ABB RobotStudio station: 00_Proyecto_RI_Irene_Perdiguero.rspag

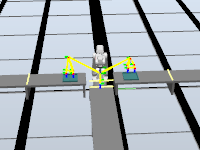
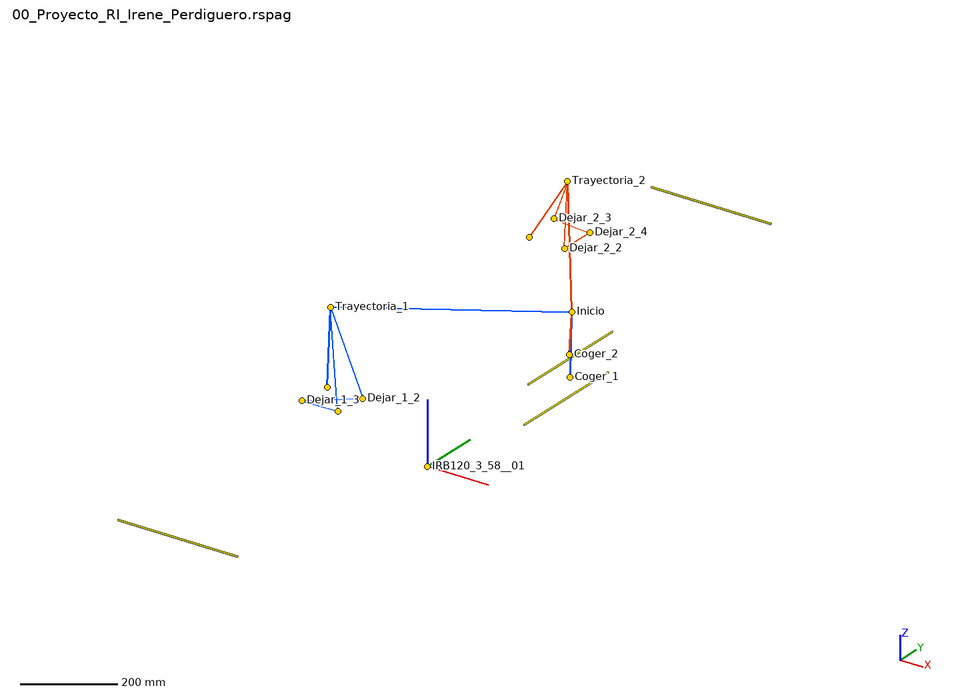
[picture v1: parts stored in the station drawn from their meshes, with robot base, taught points and paths (robot models come from the ABB library and are not in the file)]
--- station ---
Station 00_Proyecto_RI_Irene_Perdiguero (saved by RobotStudio 21.2.9526.0)
Controller Controlador1
  mechanical unit ROB_1: IRB120_3_58__01, 6 joints, base frame (0, 0, 0) mm
Layout (positions relative to the parent item):
  - IRB120_3_58__01 [mechanism, from Robots\IRB120_3_58_G_01.rslib] at (0, 0, 0) mm; joint values [-0.05, 0.292, -0.2841, -0.0016, 1.5947, -0.05] (rad or m)
  - Ventosa [mechanism, from Libraries\Ventosa.rslib] at (377.49, -19, 544.24) mm, rotated rx 180 ry -1.82 rz -180 deg
  - Producto_1 [part] at (808.06, -356.02, 0) mm, size 40 x 40 x 100 mm
  - Producto_2 [part] at (939.96, 363, 0) mm, size 40 x 39.4 x 150 mm
  - Cinta [smart component]
      signals: DI MARCHA, DI COGER_1, DI COGER_2, DI DEJAR_1, DI DEJAR_2, DO PRODUCTO_1, DO PRODUCTO_2
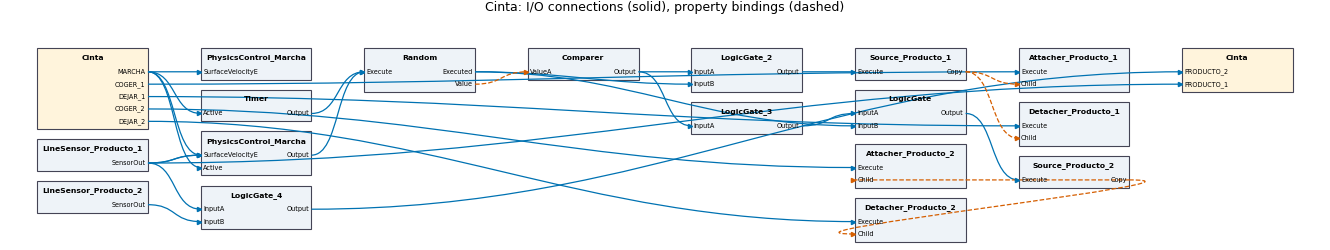
      connections:
        Cinta.MARCHA -> PhysicsControl_Marcha.SurfaceVelocityEnabled
        Cinta.MARCHA -> Timer.Active
        Timer.Output -> Random.Execute
        Comparer.Output -> LogicGate_2.InputA
        Comparer.Output -> LogicGate_3.InputA
        LogicGate_3.Output -> LogicGate.InputA
        Random.Executed -> LogicGate_2.InputB
        Random.Executed -> LogicGate.InputB
        LogicGate.Output -> Source_Producto_2.Execute
        LogicGate_2.Output -> Source_Producto_1.Execute
        LineSensor_Producto_1.SensorOut -> PhysicsControl_Paro.SurfaceVelocityEnabled
        LineSensor_Producto_1.SensorOut -> LogicGate_4.InputA
        LineSensor_Producto_2.SensorOut -> LogicGate_4.InputB
        Cinta.MARCHA -> PhysicsControl_Marcha.SurfaceVelocityEnabled
        LineSensor_Producto_1.SensorOut -> PhysicsControl_Paro.SurfaceVelocityEnabled
        Cinta.COGER_1 -> Attacher_Producto_1.Execute
        Cinta.DEJAR_1 -> Detacher_Producto_1.Execute
        Cinta.COGER_2 -> Attacher_Producto_2.Execute
        Cinta.DEJAR_2 -> Detacher_Producto_2.Execute
        Timer.Output -> Random.Execute
        Cinta.MARCHA -> Timer.Active
        LogicGate_4.Output -> Cinta.PRODUCTO_2
        LineSensor_Producto_1.SensorOut -> Cinta.PRODUCTO_1
        Random.Value => Comparer.ValueA
        Source_Producto_1.Copy => Attacher_Producto_1.Child
        Source_Producto_1.Copy => Detacher_Producto_1.Child
        Source_Producto_2.Copy => Attacher_Producto_2.Child
        Source_Producto_2.Copy => Detacher_Producto_2.Child
    - Source_Producto_1 [smart component, from Components\Source.rslib]
        properties: Source=Producto_1; Copy=(none); Parent=(none); Position=[0.8 -0.019 0.215]; Orientation=[0 0 0]; Transient=true; PhysicsBehavior=3
    - Source_Producto_2 [smart component, from Components\Source.rslib]
        properties: Source=Producto_2; Copy=(none); Parent=(none); Position=[0.8 -0.019 0.215]; Orientation=[0 0 0]; Transient=true; PhysicsBehavior=3
    - Cinta [part, from Libraries\Cinta.rslib] at (1750.47, 145.65, 0) mm, rotated rx -90 ry 0 rz 0 deg
    - LineSensor_Producto_1 [smart component, from Components\LineSensor.rslib]
        properties: Start=[0.35 0.145646 0.255]; End=[0.35 -0.154354 0.255]; Radius=0.002; SensedPart=(none); SensedPoint=[0 0 0]
      - _sensorPart_ [part], size 4 x 300 x 4 mm
    - LineSensor_Producto_2 [smart component, from Components\LineSensor.rslib]
        properties: Start=[0.36 0.145646 0.35]; End=[0.36 -0.154354 0.35]; Radius=0.002; SensedPart=(none); SensedPoint=[0 0 0]
      - _sensorPart_ [part], size 4 x 300 x 4 mm
    - Random [smart component, from Components\Random.rslib]
        properties: Value=0.495753585591797; Min=0; Max=2
    - LogicGate [smart component, from Components\LogicGate.rslib]
        properties: Operator=AND; Delay=0
    - LogicGate_2 [smart component, from Components\LogicGate.rslib]
        properties: Operator=AND; Delay=0
    - Comparer [smart component, from Components\Comparer.rslib]
        properties: ValueA=0.495753585591797; Operator=>=; ValueB=1
    - LogicGate_3 [smart component, from Components\LogicGate.rslib]
        properties: Operator=NOT; Delay=0
    - LogicGate_4 [smart component, from Components\LogicGate.rslib]
        properties: Operator=AND; Delay=0
    - PhysicsControl_Marcha [smart component, from Components\PhysicsControl.rslib]
        properties: Object=Cinta; Behavior=1; SurfaceVelocity=0.1
    - Attacher_Producto_1 [smart component, from Components\Attacher.rslib]
        properties: Parent=Ventosa; Flange=0; Child=(none); Mount=false; Offset=[0 0 0]; Orientation=[0 0 0]
    - Detacher_Producto_1 [smart component, from Components\Detacher.rslib]
        properties: Child=(none); KeepPosition=true
    - Attacher_Producto_2 [smart component, from Components\Attacher.rslib]
        properties: Parent=Ventosa; Flange=0; Child=(none); Mount=false; Offset=[0 0 0]; Orientation=[0 0 0]
    - Detacher_Producto_2 [smart component, from Components\Detacher.rslib]
        properties: Child=(none); KeepPosition=true
    - Timer [smart component, from Components\Timer.rslib]
        properties: StartTime=3.4; Interval=8; Repeat=true; CurrentTime=0
  - Cinta_1 [smart component]
      signals: DI MARCHA, DO LISTO_1
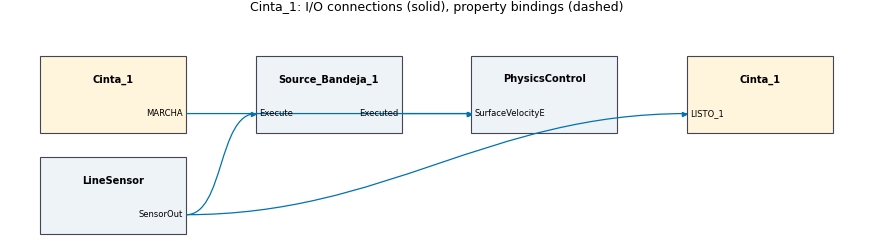
      connections:
        Cinta_1.MARCHA -> PhysicsControl.SurfaceVelocityEnabled
        LineSensor.SensorOut -> Source_Bandeja_1.Execute
        Source_Bandeja_1.Executed -> PhysicsControl.SurfaceVelocityEnabled
        LineSensor.SensorOut -> Cinta_1.LISTO_1
    - Cinta_1 [part, from Libraries\Cinta.rslib] at (192.93, -1703.86, 0) mm, rotated rx -90 ry 0 rz -90 deg
    - Positioner_Bandeja_1 [smart component, from Components\Positioner.rslib]
        properties: Object=Bandeja_1; Position=[0.043 -0.399 0.217576]; Orientation=[0 0 0]; Reference=Global; ReferenceObject=(none)
    - Bandeja_1 [part, from Libraries\Bandeja.rslib] at (43, -398.99, 216.59) mm, rotated rx 0 ry 0 rz 0.02 deg
    - PhysicsControl [smart component, from Components\PhysicsControl.rslib]
        properties: Object=Cinta_1; Behavior=1; SurfaceVelocity=0.1
    - LineSensor [smart component, from Components\LineSensor.rslib]
        properties: Start=[0.192928 -0.954267 0.23]; End=[-0.107072 -0.954267 0.23]; Radius=0.002; SensedPart=(none); SensedPoint=[0 0 0]
      - _sensorPart_ [part], size 300 x 4 x 4 mm
    - Source_Bandeja_1 [smart component, from Components\Source.rslib]
        properties: Source=Bandeja_1; Copy=(none); Parent=(none); Position=[0.043 -0.399 0.2176]; Orientation=[0 0 0]; Transient=true; PhysicsBehavior=3
  - Cinta_2 [smart component]
      signals: DI MARCHA, DO LISTO_2
      connections:
        Cinta_2.MARCHA -> PhysicsControl.SurfaceVelocityEnabled
        LineSensor_2.SensorOut -> Source_Bandeja_2.Execute
        Source_Bandeja_2.Executed -> PhysicsControl.SurfaceVelocityEnabled
        LineSensor_2.SensorOut -> Cinta_2.LISTO_2
    - Cinta_2 [part, from Libraries\Cinta.rslib] at (-103.91, 1697.08, 0) mm, rotated rx -90 ry 0 rz 90 deg
    - Positioner_Bandeja_2 [smart component, from Components\Positioner.rslib]
        properties: Object=Bandeja_2; Position=[0.046 0.408 0.217587]; Orientation=[0 0 0]; Reference=Global; ReferenceObject=(none)
    - Bandeja_2 [part, from Libraries\Bandeja.rslib] at (46, 408, 216.59) mm
    - PhysicsControl [smart component, from Components\PhysicsControl.rslib]
        properties: Object=Cinta_2; Behavior=1; SurfaceVelocity=0.1
    - LineSensor_2 [smart component, from Components\LineSensor.rslib]
        properties: Start=[0.196088 0.947493 0.23]; End=[-0.103912 0.947493 0.23]; Radius=0.002; SensedPart=(none); SensedPoint=[0 0 0]
      - _sensorPart_ [part], size 300 x 4 x 4 mm
    - Source_Bandeja_2 [smart component, from Components\Source.rslib]
        properties: Source=Bandeja_2; Copy=(none); Parent=(none); Position=[0.046 0.408 0.2176]; Orientation=[0 0 0]; Transient=true; PhysicsBehavior=3
Attachment: Ventosa is attached to IRB120_3_58__01 / Link6
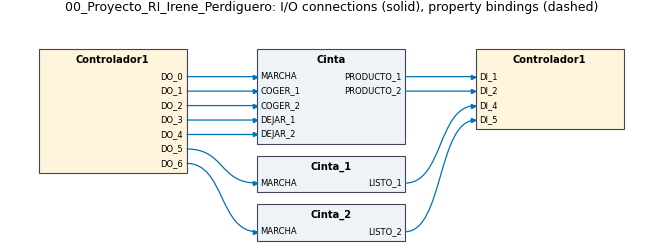
Station logic (signal -> signal, property => property):
  Controlador1.DO_0 -> Cinta.MARCHA
  Controlador1.DO_1 -> Cinta.COGER_1
  Controlador1.DO_2 -> Cinta.COGER_2
  Controlador1.DO_3 -> Cinta.DEJAR_1
  Controlador1.DO_4 -> Cinta.DEJAR_2
  Cinta.PRODUCTO_1 -> Controlador1.DI_1
  Cinta.PRODUCTO_2 -> Controlador1.DI_2
  Controlador1.DO_5 -> Cinta_1.MARCHA
  Controlador1.DO_6 -> Cinta_2.MARCHA
  Cinta_1.LISTO_1 -> Controlador1.DI_4
  Cinta_2.LISTO_2 -> Controlador1.DI_5

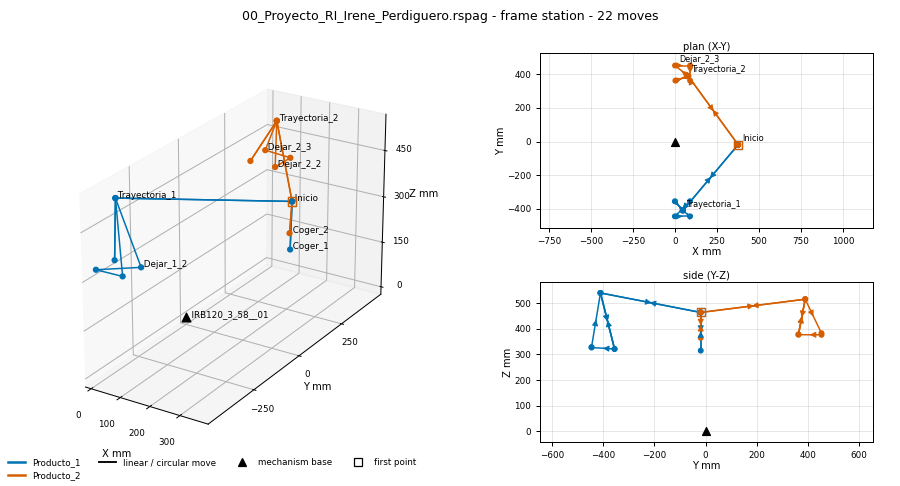
[picture p0: tool path of 00_Proyecto_RI_Irene_Perdiguero.rspag in frame station, 22 of 22 moves have a stored position in this frame; points joined in program order, loops and branches not executed]
--- Backups/Controlador1/RAPID/TASK1/PROGMOD/CalibData.mod ---
MODULE CalibData
    PERS tooldata Ventosa:=[TRUE,[[0,0,80],[1,0,0,0]],[0.1,[0,0,1],[1,0,0,0],0,0,0]];
    TASK PERS wobjdata Entorno:=[FALSE,TRUE,"",[[0,0,0],[1,0,0,0]],[[0,0,0],[1,0,0,0]]];
ENDMODULE

--- Backups/Controlador1/RAPID/TASK1/PROGMOD/Module1.mod ---
MODULE Module1
    CONST robtarget Trayectoria_Dejar_1:=[[-2.131996898,-355.446793269,459.714373735],[0.002016963,0.999256804,0.038491712,0.000399842],[-2,0,0,0],[9E+09,9E+09,9E+09,9E+09,9E+09,9E+09]];
    CONST robtarget Dejar_Producto_1:=[[-2.131996806,-355.446806361,459.714425121],[0.002016983,0.999256804,0.038491713,0.000399841],[-2,0,0,0],[9E+09,9E+09,9E+09,9E+09,9E+09,9E+09]];
    CONST robtarget Inicio:=[[374.939892389,-18.999999171,464.275766351],[0.015920536,0.000000001,-0.99987326,-0.000000001],[-1,-1,-1,0],[9E+09,9E+09,9E+09,9E+09,9E+09,9E+09]];
    CONST robtarget Coger_1:=[[370.192,-19,315],[0.006807824,0,0.999976827,0],[0,0,0,0],[9E+09,9E+09,9E+09,9E+09,9E+09,9E+09]];
    CONST robtarget Trayectoria_1:=[[45.337309364,-411.041582777,540.541875459],[0.002016947,0.999256807,0.03849163,0.000399844],[-1,0,1,0],[9E+09,9E+09,9E+09,9E+09,9E+09,9E+09]];
    CONST robtarget Dejar_1:=[[-2.005,-355.983,321.539],[0.00345143,-0.999994044,0,0],[0,0,0,0],[9E+09,9E+09,9E+09,9E+09,9E+09,9E+09]];
    CONST robtarget Coger_2:=[[367.753,-19.249,365],[0.011265611,0,-0.999936541,0],[0,0,0,0],[9E+09,9E+09,9E+09,9E+09,9E+09,9E+09]];
    CONST robtarget Trayectoria_2:=[[77.890283908,389.307652093,515.990648683],[0.006482552,-0.999978988,-0.000000115,-0.000000006],[0,0,-2,0],[9E+09,9E+09,9E+09,9E+09,9E+09,9E+09]];
    CONST robtarget Dejar_2:=[[0.999979445,363.000009526,378.395460462],[0.00678485,-0.999976983,-0.000000007,0],[0,0,-2,0],[9E+09,9E+09,9E+09,9E+09,9E+09,9E+09]];
    CONST robtarget Dejar_1_2:=[[88,-356.02,321.348],[0.00345143,-0.999994044,0,0],[-1,0,1,0],[9E+09,9E+09,9E+09,9E+09,9E+09,9E+09]];
    CONST robtarget Dejar_1_3:=[[-1.999973838,-446.020008039,327.099676047],[0.003451442,-0.999994044,-0.000000033,0],[-2,-1,0,0],[9E+09,9E+09,9E+09,9E+09,9E+09,9E+09]];
    CONST robtarget Dejar_1_4:=[[87.999978489,-446.020020044,328.84303757],[0.003451441,-0.999994044,0.000000036,0.000000002],[-1,0,1,0],[9E+09,9E+09,9E+09,9E+09,9E+09,9E+09]];
    CONST robtarget Dejar_2_2:=[[88.999994314,362.995017557,377.328653121],[0.00678489,-0.999976982,-0.00000003,-0.000000005],[0,0,-2,0],[9E+09,9E+09,9E+09,9E+09,9E+09,9E+09]];
    CONST robtarget Dejar_2_3:=[[-0.999989304,453.00001379,383.168859939],[0.006784829,-0.999976983,-0.000000016,0],[1,-1,-1,0],[9E+09,9E+09,9E+09,9E+09,9E+09,9E+09]];
    CONST robtarget Dejar_2_4:=[[89.000011483,453.000019118,376.887455285],[0.006784875,-0.999976982,-0.000000017,-0.000000002],[0,0,-2,0],[9E+09,9E+09,9E+09,9E+09,9E+09,9E+09]];
    VAR num cont_1:=0;
    VAR num cont_2:=0;

    !***********************************************************
    !
    ! Módulo:  Module1
    !
    ! Descripción:
    !   Paletizado de dos tipos de productos: un cubo bajo y un cilindro alto.
    !   Se almacenarán 4 cubos sobre el palet de la cinta 1 y 4 cilindros sobre el palet de la cinta 2
    !   Cuando los palet estén llenos la cinta transportadora se pone en marcha y cuando esté a la mitad del recorrido un pallet nuevo aparece y repetimos la misma operación
    ! Autor: Irene Perdiguero Gómez
    !
    ! Versión: 1.0
    !
    !***********************************************************


    !***********************************************************
    !
    ! Procedimiento Main
    !
    !   Este es el punto de entrada de su programa
    !
    !***********************************************************
    PROC main()
!        Hago que una entrada me ponga todas las salidas a 0
        IF DI_3=1 THEN
            Reset DO_0;
            Reset DO_1;
            Reset DO_2;
            Reset DO_3;
            Reset DO_4;
            Reset DO_5;
            Reset DO_6;
        ENDIF

!        Simulamos un pulsador de marcha para que comience la cinta transportadora a moverse y a salir los elementos
        IF DI_0 = 1 THEN
            SetDO DO_0,1;
        ENDIF

!        Si detecta el producto uno (el cubo bajo), va al path del producto 1 y para la cinta transportadora
        IF DI_1 = 1 and DI_2 = 0 THEN
            SetDO DO_0,0;
            Producto_1;
        ENDIF

!        Si detecta el producto dos (el cilindro alto), va al path del producto 2 y para la cinta transportadora
        IF DI_2 = 1 and DI_1 = 1 THEN
            SetDO DO_0,0;
            Producto_2;
        ENDIF

    ENDPROC

    PROC Producto_1()
        MoveL Inicio,v500,fine,Ventosa\WObj:=Entorno;
        MoveL Coger_1,v500,fine,Ventosa\WObj:=Entorno;
!        Activamos ventosa, cogemos el producto y ponemos en marcha la cinta transportadora
        SetDO DO_1,1;
        WaitTime 0.5;
        SetDO DO_0,1;
        MoveL Inicio,v500,fine,Ventosa\WObj:=Entorno;
        MoveL Trayectoria_1,v500,fine,Ventosa\WObj:=Entorno;
!        He programado una posicion por cada sitio donde tiene que dejarlo
        IF cont_1=1 THEN
             MoveL Dejar_1_2,v1000,fine,Ventosa\WObj:=Entorno;
        ENDIF
        IF cont_1=2 THEN
             MoveL Dejar_1_3,v1000,fine,Ventosa\WObj:=Entorno;
        ENDIF
        IF cont_1=3 THEN
             MoveL Dejar_1_4,v1000,fine,Ventosa\WObj:=Entorno;
             WaitTime 0.5;
             SetDO DO_1,0;
             SetDO DO_3,1;
             MoveL Trayectoria_1,v500,fine,Ventosa\WObj:=Entorno;
             SetDO DO_5,1;
        ENDIF
!        Cuando este lleno el palet ponemos el contador a cero para cuando llegue el nuevo palet hacer lo mismo
        IF cont_1=4 THEN
            cont_1:=0;
        ENDIF
        IF cont_1=0 THEN
             MoveL Dejar_1,v1000,fine,Ventosa\WObj:=Entorno;
        ENDIF
        WaitTime 0.5;
!        Desactivamos salida que utilizamos para coger y activamos la de dejar
        SetDO DO_1,0;
        SetDO DO_3,1;
        MoveL Trayectoria_1,v500,fine,Ventosa\WObj:=Entorno;
        MoveL Inicio,v500,fine,Ventosa\WObj:=Entorno;
!        Desactivamos la salida que utilizamos para dejar
        SetDO DO_3,0;
        IF DI_4 = 1 and cont_1 = 0 THEN
            WaitTime 3;
            Reset DO_5;
        ENDIF
!        Contador de cuantos elementos lleva colocados
        cont_1:=cont_1+1;

    ENDPROC
    PROC Producto_2()
        MoveL Inicio,v500,fine,Ventosa\WObj:=Entorno;
        MoveL Coger_2,v500,fine,Ventosa\WObj:=Entorno;
!        Activamos ventosa, cogemos el producto y ponemos en marcha la cinta transportadora
        SetDO DO_2,1;
        WaitTime 0.5;
        SetDO DO_0,1;
        MoveL Inicio,v500,fine,Ventosa\WObj:=Entorno;
        MoveL Trayectoria_2,v500,fine,Ventosa\WObj:=Entorno;
!        He programado una posicion por cada sitio donde tiene que dejarlo
        IF cont_2=1 THEN
             MoveL Dejar_2_3,v1000,fine,Ventosa\WObj:=Entorno;
        ENDIF
        IF cont_2=2 THEN
             MoveL Dejar_2_4,v1000,fine,Ventosa\WObj:=Entorno;
        ENDIF
        IF cont_2=3 THEN
             MoveL Dejar_2_2,v1000,fine,Ventosa\WObj:=Entorno;
             WaitTime 0.5;
             SetDO DO_2,0;
             SetDO DO_4,1;
             MoveL Trayectoria_2,v500,fine,Ventosa\WObj:=Entorno;
             Set DO_6;
        ENDIF
!        Cuando este lleno el palet ponemos el contador a cero para cuando llegue el nuevo palet hacer lo mismo
        IF cont_2=4 THEN
            cont_2:=0;
        ENDIF
        IF cont_2=0 THEN
             MoveL Dejar_2,v1000,fine,Ventosa\WObj:=Entorno;
        ENDIF
        WaitTime 0.5;
!         Desactivamos salida que utilizamos para coger y activamos la de dejar
        SetDO DO_2,0;
        SetDO DO_4,1;
        MoveL Trayectoria_2,v500,fine,Ventosa\WObj:=Entorno;
        MoveL Inicio,v500,fine,Ventosa\WObj:=Entorno;
!        Desactivamos la salida que utilizamos para dejar
        SetDO DO_4,0;
        IF DI_5 = 1 and cont_2 = 0 THEN
            WaitTime 3;
            Reset DO_6;
        ENDIF
!        Contador de cuantos elementos lleva colocados
        cont_2:=cont_2+1;

    ENDPROC
ENDMODULE

--- Backups/Controlador1/SYSPAR/EIO.cfg ---
EIO:CFG_1.0:6:1::
#
INDUSTRIAL_NETWORK:

      -Name "DeviceNet" -Label "DeviceNet Master/Slave Network" -Address "2"
#
DEVICENET_DEVICE:

      -Name "d652" -VendorName "ABB Robotics" -ProductName "24 VDC I/O Device"\
      -Label "DSQC 652 24 VDC I/O Device" -Address 10 -ProductCode 26\
      -DeviceType 7 -ConnectionType "COS" -OutputSize 2 -InputSize 2
#
DEVICENET_INTERNAL_DEVICE:

      -Name "DN_Internal_Device" -VendorName "ABB Robotics"\
      -ProductName "DeviceNet Internal Slave Device"
#
EIO_SIGNAL:

      -Name "DI_0" -SignalType "DI" -Device "d652" -DeviceMap "0"

      -Name "DI_1" -SignalType "DI" -Device "d652" -DeviceMap "1"

      -Name "DI_2" -SignalType "DI" -Device "d652" -DeviceMap "2"

      -Name "DI_3" -SignalType "DI" -Device "d652" -DeviceMap "3"

      -Name "DI_4" -SignalType "DI" -Device "d652" -DeviceMap "4"

      -Name "DI_5" -SignalType "DI" -Device "d652" -DeviceMap "5"

      -Name "DO_0" -SignalType "DO" -Device "d652" -DeviceMap "0"

      -Name "DO_1" -SignalType "DO" -Device "d652" -DeviceMap "1"

      -Name "DO_2" -SignalType "DO" -Device "d652" -DeviceMap "2"

      -Name "DO_3" -SignalType "DO" -Device "d652" -DeviceMap "3"

      -Name "DO_4" -SignalType "DO" -Device "d652" -DeviceMap "4"

      -Name "DO_5" -SignalType "DO" -Device "d652" -DeviceMap "5"

      -Name "DO_6" -SignalType "DO" -Device "d652" -DeviceMap "6"
